# B&R Automation Studio project CombinedLinenSoiledA9KAN (part 18)

#### _actIFCmd.st
```iecst
(********************************************************************
 * COPYRIGHT -- Herbert Kannegiesser GmbH
 ********************************************************************
 * Program: svCPCache
 * File: _actIFCmd.st
 * Author: hunholz
 * Created: March 30, 2012
 ********************************************************************
 * Implementation of program svCPCache
 ********************************************************************)

(* Add a new action to your IEC program or library *)
ACTION _actIFCmd:

	CASE _enCmd OF

		cs_CmdIdle:

		// Warte auf Kommando

			CASE IFsvCPCache.In.wCmd OF

				KG_CMD_NOCOMMAND:

					IFsvCPCache.Out.wCmdResponse := KG_CMD_NOCOMMAND;

				SVCPCACHE_CMD_GETPROG:

					IFsvCPCache.Out.rRespSoilFactor 		:= 1.0;
					IFsvCPCache.Out.utfRespCategoryName		:= "";
					IFsvCPCache.Out.wRespColidxBack			:= 15;
					IFsvCPCache.Out.wRespColidxFor			:= 1;
					IFsvCPCache.Out.wRespLoadrate			:= 100;
					IFsvCPCache.Out.wRespProgramNo			:= 0;
					IFsvCPCache.Out.utfRespProgramName		:= "";

					IFsvCPCache.Out.wRespFromDB				:= SVCPCACHE_DBREQ_LOCAL;

					_TrimCat(sCategory := IFsvCPCache.In.sReqCategory);
					_sCategory := _TrimCat.sOutCategory;

					IF _sCategory <> '' THEN

						// Suche Kategorie auf jeden Fall lokal

						_xCategoryExist := FALSE;
						_wCategoryIdx := 0;

						FOR _i := 1 TO SVCPCACHE_CNT_RELATIONS DO

							IF _CPCache[_i].dtTimeStamp = USINT_TO_DT(0) THEN
								EXIT;
							ELSIF _CPCache[_i].sCategory = _sCategory THEN
								_xCategoryExist := TRUE;
								_wCategoryIdx := _i;
								EXIT;
							END_IF

						END_FOR

						// Entscheidung, ob in der Datenbank gesucht werden soll

						IF IFsvCPCache.In.wReqUseDB = SVCPCACHE_DBREQ_LOCAL THEN

							IF _xCategoryExist THEN

								IFsvCPCache.Out.rRespSoilFactor 		:= _CPCache[_wCategoryIdx].rSoilfactor;
								IFsvCPCache.Out.utfRespCategoryName		:= _CPCache[_wCategoryIdx].utfCategoryName;
								IFsvCPCache.Out.wRespColidxBack			:= _CPCache[_wCategoryIdx].wColBack;
								IFsvCPCache.Out.wRespColidxFor			:= _CPCache[_wCategoryIdx].wColFor;
								IFsvCPCache.Out.wRespLoadrate			:= _CPCache[_wCategoryIdx].wLoadrate;
								IFsvCPCache.Out.wRespProgramNo			:= _CPCache[_wCategoryIdx].wProgramNo;

								FOR _i := 1 TO IFmnParam.Out.Edit.wCntNamelist DO

									IF IFmnParam.Out.Edit.wNameListNo[_i] = IFsvCPCache.Out.wRespProgramNo THEN
										IFsvCPCache.Out.utfRespProgramName := IFmnParam.Out.Edit.utfNameListName[_i];
										EXIT;
									END_IF

								END_FOR

								IFsvCPCache.Out.wCmdResponse := SVCPCACHE_CMD_GETPROG;
								_enCmd := cs_CmdWaitForNoCommand;

							ELSE

								IFsvCPCache.Out.wCmdResponse := SVCPCACHE_STAT_CATEGORYNOTEXIST;
								_enCmd := cs_CmdWaitForNoCommand;

							END_IF

						ELSE // Abfrage der Datenbank starten

							IF IFhlDFII.Out.xConnected THEN

								IFsvCPCache.Out.wCmdResponse := KG_STAT_BUSY;
								_enCmd := cs_CmdWaitForDB;

							ELSE

								IFsvCPCache.Out.wCmdResponse := SVCPCACHE_STAT_DBNOTREADY;
								_enCmd := cs_CmdWaitForNoCommand;

								IF _xCategoryExist THEN

									IFsvCPCache.Out.rRespSoilFactor 		:= _CPCache[_wCategoryIdx].rSoilfactor;
									IFsvCPCache.Out.utfRespCategoryName		:= _CPCache[_wCategoryIdx].utfCategoryName;
									IFsvCPCache.Out.wRespColidxBack			:= _CPCache[_wCategoryIdx].wColBack;
									IFsvCPCache.Out.wRespColidxFor			:= _CPCache[_wCategoryIdx].wColFor;
									IFsvCPCache.Out.wRespLoadrate			:= _CPCache[_wCategoryIdx].wLoadrate;
									IFsvCPCache.Out.wRespProgramNo			:= _CPCache[_wCategoryIdx].wProgramNo;

									FOR _i := 1 TO IFmnParam.Out.Edit.wCntNamelist DO

										IF IFmnParam.Out.Edit.wNameListNo[_i] = IFsvCPCache.Out.wRespProgramNo THEN
											IFsvCPCache.Out.utfRespProgramName := IFmnParam.Out.Edit.utfNameListName[_i];
											EXIT;
										END_IF

									END_FOR

								END_IF

							END_IF

						END_IF

					ELSE

						IFsvCPCache.Out.wCmdResponse := SVCPCACHE_STAT_INVALIDCATEGORY;
						_enCmd := cs_CmdWaitForNoCommand;

					END_IF

				SVCPCACHE_CMD_INSERTCATEGORY:

					_wCmd := SVCPCACHE_CMD_INSERTCATEGORY;

					IF IFsvCPCache.Out.wCntRelations < SVCPCACHE_CNT_RELATIONS THEN

						_TrimCat(sCategory := IFsvCPCache.In.sReqCategory);
						_sCategory := _TrimCat.sOutCategory;

						IF _sCategory <> '' THEN

							_xCategoryExist := FALSE;

							FOR _i := 1 TO SVCPCACHE_CNT_RELATIONS DO

								IF _CPCache[_i].dtTimeStamp = USINT_TO_DT(0) THEN
									EXIT;
								ELSIF _CPCache[_i].sCategory = _sCategory THEN
									_xCategoryExist := TRUE;
									EXIT;
								END_IF

							END_FOR

							IF NOT _xCategoryExist THEN

								_DTGetTime(enable := TRUE);

								FOR _i := 1 TO SVCPCACHE_CNT_RELATIONS DO

									IF _CPCache[_i].dtTimeStamp = USINT_TO_DT(0) THEN

										_CPCache[_i].dtTimeStamp := _DTGetTime.DT1;
										_CPCache[_i].sCategory := _sCategory;
										_CPCache[_i].utfCategoryName := IFsvCPCache.In.utfReqCategoryName;
										_CPCache[_i].wProgramNo := IFsvCPCache.In.wReqProgramNo;
										_CPCache[_i].rSoilfactor := IFsvCPCache.In.rReqSoilfactor;
										_CPCache[_i].wLoadrate := IFsvCPCache.In.wReqLoadrate;
										_CPCache[_i].wColFor := IFsvCPCache.In.wReqColidxFor;
										_CPCache[_i].wColBack := IFsvCPCache.In.wReqColidxBack;

										IFsvCPCache.Out.wCntRelations := IFsvCPCache.Out.wCntRelations + 1;

										EXIT;

									ELSIF brsstrcmp(ADR(_CPCache[_i].sCategory),ADR(_sCategory)) > 0 THEN

										brsmemmove(ADR(_CPCache[_i+1]), ADR(_CPCache[_i]), SIZEOF(_CPCache[1])*(IFsvCPCache.Out.wCntRelations-_i+1) );

										_CPCache[_i].dtTimeStamp := _DTGetTime.DT1;
										_CPCache[_i].sCategory := _sCategory;
										_CPCache[_i].utfCategoryName := IFsvCPCache.In.utfReqCategoryName;
										_CPCache[_i].wProgramNo := IFsvCPCache.In.wReqProgramNo;
										_CPCache[_i].rSoilfactor := IFsvCPCache.In.rReqSoilfactor;
										_CPCache[_i].wLoadrate := IFsvCPCache.In.wReqLoadrate;
										_CPCache[_i].wColFor := IFsvCPCache.In.wReqColidxFor;
										_CPCache[_i].wColBack := IFsvCPCache.In.wReqColidxBack;

										IFsvCPCache.Out.wCntRelations := IFsvCPCache.Out.wCntRelations + 1;

										EXIT;

									END_IF

								END_FOR

								_enSave := cs_SaveCreateCSV;

								_enCmd := cs_CmdSave;

							ELSE

								IFsvCPCache.Out.wCmdResponse := SVCPCACHE_STAT_CATEGORYEXIST;
								_enCmd := cs_CmdWaitForNoCommand;

							END_IF

						ELSE

							IFsvCPCache.Out.wCmdResponse := SVCPCACHE_STAT_INVALIDCATEGORY;
							_enCmd := cs_CmdWaitForNoCommand;

						END_IF

					ELSE

						IFsvCPCache.Out.wCmdResponse := SVCPCACHE_STAT_NOSPACE;
						_enCmd := cs_CmdWaitForNoCommand;

					END_IF

				SVCPCACHE_CMD_UPDATECATEGORY:

					_wCmd := SVCPCACHE_CMD_UPDATECATEGORY;

					IF IFsvCPCache.Out.wCntRelations > 0 THEN

						_TrimCat(sCategory := IFsvCPCache.In.sReqCategory);
						_sCategory := _TrimCat.sOutCategory;

						IF _sCategory <> '' THEN

							_xCategoryExist := FALSE;

							FOR _i := 1 TO SVCPCACHE_CNT_RELATIONS DO

								IF _CPCache[_i].dtTimeStamp = USINT_TO_DT(0) THEN
									EXIT;
								ELSIF _CPCache[_i].sCategory = _sCategory THEN
									_xCategoryExist := TRUE;
									EXIT;
								END_IF

							END_FOR

							IF _xCategoryExist THEN

								_DTGetTime(enable := TRUE);

								_CPCache[_i].dtTimeStamp := _DTGetTime.DT1;
								_CPCache[_i].sCategory := _sCategory;
								_CPCache[_i].utfCategoryName := IFsvCPCache.In.utfReqCategoryName;
								_CPCache[_i].wProgramNo := IFsvCPCache.In.wReqProgramNo;
								_CPCache[_i].rSoilfactor := IFsvCPCache.In.rReqSoilfactor;
								_CPCache[_i].wLoadrate := IFsvCPCache.In.wReqLoadrate;
								_CPCache[_i].wColFor := IFsvCPCache.In.wReqColidxFor;
								_CPCache[_i].wColBack := IFsvCPCache.In.wReqColidxBack;

								_enSave := cs_SaveCreateCSV;

								_enCmd := cs_CmdSave;

							ELSE

								IFsvCPCache.Out.wCmdResponse := SVCPCACHE_STAT_CATEGORYNOTEXIST;
								_enCmd := cs_CmdWaitForNoCommand;

							END_IF

						ELSE

							IFsvCPCache.Out.wCmdResponse := SVCPCACHE_STAT_INVALIDCATEGORY;
							_enCmd := cs_CmdWaitForNoCommand;

						END_IF

					ELSE

						IFsvCPCache.Out.wCmdResponse := SVCPCACHE_STAT_CATEGORYLISTEMPTY;
						_enCmd := cs_CmdWaitForNoCommand;

					END_IF

				SVCPCACHE_CMD_DELETECATEGORY:

					_wCmd := SVCPCACHE_CMD_DELETECATEGORY;

					IF IFsvCPCache.Out.wCntRelations > 0 THEN

						_TrimCat(sCategory := IFsvCPCache.In.sReqCategory);
						_sCategory := _TrimCat.sOutCategory;

						IF _sCategory <> '' THEN

							_xCategoryExist := FALSE;

							FOR _i := 1 TO SVCPCACHE_CNT_RELATIONS DO

								IF _CPCache[_i].dtTimeStamp = USINT_TO_DT(0) THEN
									EXIT;
								ELSIF _CPCache[_i].sCategory = _sCategory THEN
									_xCategoryExist := TRUE;
									EXIT;
								END_IF

							END_FOR

							IF _xCategoryExist THEN

								IF _i < IFsvCPCache.Out.wCntRelations THEN

									brsmemmove(ADR(_CPCache[_i]), ADR(_CPCache[_i+1]), SIZEOF(_CPCache[1])*(IFsvCPCache.Out.wCntRelations-_i) );

								END_IF

								brsmemset(ADR(_CPCache[IFsvCPCache.Out.wCntRelations]), 0, SIZEOF(_CPCache[1]));

								IFsvCPCache.Out.wCntRelations := IFsvCPCache.Out.wCntRelations - 1;

								_enSave := cs_SaveCreateCSV;

								_enCmd := cs_CmdSave;

							ELSE

								IFsvCPCache.Out.wCmdResponse := SVCPCACHE_STAT_CATEGORYNOTEXIST;
								_enCmd := cs_CmdWaitForNoCommand;

							END_IF

						ELSE

							IFsvCPCache.Out.wCmdResponse := SVCPCACHE_STAT_INVALIDCATEGORY;
							_enCmd := cs_CmdWaitForNoCommand;

						END_IF

					ELSE

						IFsvCPCache.Out.wCmdResponse := SVCPCACHE_STAT_CATEGORYLISTEMPTY;
						_enCmd := cs_CmdWaitForNoCommand;

					END_IF

				SVCPCACHE_CMD_SETOFFSET:

					IFsvCPCache.Out.wListOffset := IFsvCPCache.In.wSetOffset;
					_actFillCPList;

					IFsvCPCache.Out.wCmdResponse := SVCPCACHE_CMD_SETOFFSET;
					_enCmd := cs_CmdWaitForNoCommand;

				ELSE

					IFsvCPCache.Out.wCmdResponse := KG_CMDSTAT_NOTVALID;
					_enCmd := cs_CmdWaitForNoCommand;

			END_CASE

		cs_CmdSave:

			IF _enSave = cs_SaveRdySuccess THEN

				_actFillCPList;

				IFsvCPCache.Out.wCmdResponse := _wCmd;
				_enCmd := cs_CmdWaitForNoCommand;

			ELSIF _enSave = cs_SaveRdyFault THEN

				IFsvCPCache.Out.wCmdResponse := _wSaveCSVstatus;
				_enCmd := cs_CmdWaitForNoCommand;

			END_IF

		cs_CmdWaitForDB:

			IF IFhlDFII.In.ReqProgByCat.wRequest = 0 AND IFhlDFII.Out.RespProgByCat.wResponse = 0 THEN

				IFhlDFII.In.ReqProgByCat.sCategoryNo_In := IFsvCPCache.In.sReqCategory;
				IFhlDFII.In.ReqProgByCat.wRequest		:= 2;

			ELSIF IFhlDFII.In.ReqProgByCat.wRequest = 2 AND IFhlDFII.Out.RespProgByCat.wResponse = 2 THEN

				_DTGetTime(enable := TRUE);

				IFsvCPCache.Out.rRespSoilFactor 		:= IFhlDFII.Out.RespProgByCat.rSoilfactor;
				IFsvCPCache.Out.utfRespCategoryName 	:= STRING_TO_WSTRING(IFhlDFII.Out.RespProgByCat.sCategoryName);
				IFsvCPCache.Out.wRespColidxBack			:= IFhlDFII.Out.RespProgByCat.wColorIdxBack;
				IFsvCPCache.Out.wRespColidxFor			:= IFhlDFII.Out.RespProgByCat.wColorIdxFor;
				IFsvCPCache.Out.wRespLoadrate			:= IFhlDFII.Out.RespProgByCat.wLoadrate;
				IFsvCPCache.Out.wRespProgramNo			:= IFhlDFII.Out.RespProgByCat.bProgramNo;

				FOR _i := 1 TO IFmnParam.Out.Edit.wCntNamelist DO

					IF IFmnParam.Out.Edit.wNameListNo[_i] = IFsvCPCache.Out.wRespProgramNo THEN
						IFsvCPCache.Out.utfRespProgramName := IFmnParam.Out.Edit.utfNameListName[_i];
						EXIT;
					END_IF

				END_FOR

				IFsvCPCache.Out.wRespFromDB				:= SVCPCACHE_DBREQ_DFII;

				IF _xCategoryExist AND
					_CPCache[_wCategoryIdx].utfCategoryName = IFsvCPCache.Out.utfRespCategoryName AND
					_CPCache[_wCategoryIdx].rSoilfactor = IFsvCPCache.Out.rRespSoilFactor AND
					_CPCache[_wCategoryIdx].wLoadrate = IFsvCPCache.Out.wRespLoadrate AND
					_CPCache[_wCategoryIdx].wColBack = IFsvCPCache.Out.wRespColidxBack AND
					_CPCache[_wCategoryIdx].wColFor = IFsvCPCache.Out.wRespColidxFor AND
					_CPCache[_wCategoryIdx].wProgramNo =  IFsvCPCache.Out.wRespProgramNo THEN

					// Lokale Daten sind gleich den Daten aus der Datenbank

					IFsvCPCache.Out.wCmdResponse			:= SVCPCACHE_CMD_GETPROG;
					_enCmd := cs_CmdWaitForNoCommand;

				ELSIF _xCategoryExist THEN

					// Lokale Daten werden aktualisiert

					_CPCache[_wCategoryIdx].utfCategoryName := STRING_TO_WSTRING(IFhlDFII.Out.RespProgByCat.sCategoryName);
					_CPCache[_wCategoryIdx].rSoilfactor 	:= IFhlDFII.Out.RespProgByCat.rSoilfactor;
					_CPCache[_wCategoryIdx].wLoadrate 		:= IFhlDFII.Out.RespProgByCat.wLoadrate;
					_CPCache[_wCategoryIdx].wColBack 		:= IFhlDFII.Out.RespProgByCat.wColorIdxBack;
					_CPCache[_wCategoryIdx].wColFor 		:= IFhlDFII.Out.RespProgByCat.wColorIdxFor;
					_CPCache[_wCategoryIdx].wProgramNo 		:= IFhlDFII.Out.RespProgByCat.bProgramNo;
					_CPCache[_wCategoryIdx].dtTimeStamp		:= _DTGetTime.DT1;

					_wCmd := SVCPCACHE_CMD_GETPROG;
					_enSave := cs_SaveCreateCSV;
					_enCmd := cs_CmdSave;

				ELSE

					// Es wird versucht eine neue Kategorie in den lokalen Speicher abzulegen

					IF IFsvCPCache.Out.wCntRelations < SVCPCACHE_CNT_RELATIONS THEN

						FOR _i := 1 TO SVCPCACHE_CNT_RELATIONS DO

							IF _CPCache[_i].dtTimeStamp = USINT_TO_DT(0) THEN

								_CPCache[_i].dtTimeStamp 		:= _DTGetTime.DT1;
								_CPCache[_i].sCategory 			:= _sCategory;
								_CPCache[_i].utfCategoryName 	:= STRING_TO_WSTRING(IFhlDFII.Out.RespProgByCat.sCategoryName);
								_CPCache[_i].wProgramNo 		:= IFhlDFII.Out.RespProgByCat.bProgramNo;
								_CPCache[_i].rSoilfactor 		:= IFhlDFII.Out.RespProgByCat.rSoilfactor;
								_CPCache[_i].wLoadrate 			:= IFhlDFII.Out.RespProgByCat.wLoadrate;
								_CPCache[_i].wColFor 			:= IFhlDFII.Out.RespProgByCat.wColorIdxFor;
								_CPCache[_i].wColBack 			:= IFhlDFII.Out.RespProgByCat.wColorIdxBack;

								IFsvCPCache.Out.wCntRelations := IFsvCPCache.Out.wCntRelations + 1;

								EXIT;

							ELSIF brsstrcmp(ADR(_CPCache[_i].sCategory),ADR(_sCategory)) > 0 THEN

								brsmemmove(ADR(_CPCache[_i+1]), ADR(_CPCache[_i]), SIZEOF(_CPCache[1])*(IFsvCPCache.Out.wCntRelations-_i+1) );

								_CPCache[_i].dtTimeStamp 		:= _DTGetTime.DT1;
								_CPCache[_i].sCategory 			:= _sCategory;
								_CPCache[_i].utfCategoryName 	:= STRING_TO_WSTRING(IFhlDFII.Out.RespProgByCat.sCategoryName);
								_CPCache[_i].wProgramNo 		:= IFhlDFII.Out.RespProgByCat.bProgramNo;
								_CPCache[_i].rSoilfactor 		:= IFhlDFII.Out.RespProgByCat.rSoilfactor;
								_CPCache[_i].wLoadrate 			:= IFhlDFII.Out.RespProgByCat.wLoadrate;
								_CPCache[_i].wColFor 			:= IFhlDFII.Out.RespProgByCat.wColorIdxFor;
								_CPCache[_i].wColBack 			:= IFhlDFII.Out.RespProgByCat.wColorIdxBack;

								IFsvCPCache.Out.wCntRelations := IFsvCPCache.Out.wCntRelations + 1;

								EXIT;

							END_IF

						END_FOR

						_wCmd := SVCPCACHE_CMD_GETPROG;
						_enSave := cs_SaveCreateCSV;
						_enCmd := cs_CmdSave;

					ELSE

						// Kein Platz für eine neue Kategorie

						IFsvCPCache.Out.wCmdResponse			:= SVCPCACHE_CMD_GETPROG;
						_enCmd := cs_CmdWaitForNoCommand;

					END_IF

				END_IF

				IFhlDFII.In.ReqProgByCat.wRequest		:= 0;

			ELSIF IFhlDFII.In.ReqProgByCat.wRequest = 2 AND IFhlDFII.Out.RespProgByCat.wResponse <> 65535 AND IFhlDFII.Out.RespProgByCat.wResponse <> 0 THEN

				IF _xCategoryExist THEN

					IFsvCPCache.Out.rRespSoilFactor 		:= _CPCache[_wCategoryIdx].rSoilfactor;
					IFsvCPCache.Out.utfRespCategoryName		:= _CPCache[_wCategoryIdx].utfCategoryName;
					IFsvCPCache.Out.wRespColidxBack			:= _CPCache[_wCategoryIdx].wColBack;
					IFsvCPCache.Out.wRespColidxFor			:= _CPCache[_wCategoryIdx].wColFor;
					IFsvCPCache.Out.wRespLoadrate			:= _CPCache[_wCategoryIdx].wLoadrate;
					IFsvCPCache.Out.wRespProgramNo			:= _CPCache[_wCategoryIdx].wProgramNo;

					FOR _i := 1 TO IFmnParam.Out.Edit.wCntNamelist DO

						IF IFmnParam.Out.Edit.wNameListNo[_i] = IFsvCPCache.Out.wRespProgramNo THEN
							IFsvCPCache.Out.utfRespProgramName := IFmnParam.Out.Edit.utfNameListName[_i];
							EXIT;
						END_IF

					END_FOR

					IFsvCPCache.Out.wCmdResponse 			:= SVCPCACHE_CMD_GETPROG;

				ELSE

					IFsvCPCache.Out.wCmdResponse			:= IFhlDFII.Out.RespProgByCat.wResponse;

				END_IF

				IFhlDFII.In.ReqProgByCat.wRequest		:= 0;
				_enCmd := cs_CmdWaitForNoCommand;

			END_IF

		cs_CmdWaitForNoCommand:

			IF IFsvCPCache.In.wCmd = KG_CMD_NOCOMMAND THEN

				IFsvCPCache.Out.wCmdResponse := KG_STAT_OK;

				_enCmd := cs_CmdIdle;

			END_IF

	END_CASE

END_ACTION
```

#### _actSaveCSV.st
```iecst
(********************************************************************
 * COPYRIGHT -- Herbert Kannegiesser GmbH
 ********************************************************************
 * Program: svCPCache
 * File: _actSaveCSV.st
 * Author: hunholz
 * Created: March 30, 2012
 ********************************************************************
 * Implementation of program svCPCache
 ********************************************************************)

(* Schrittkette zum Speichern der Kategorie-Programm-Zuordnung *)
ACTION _actSaveCSV:

	_wSaveCSVstatus := ERR_OK;

	CASE _enSave OF

		cs_SaveIdle:

			// Tue nichts

		cs_SaveCreateCSV:

			_SaveMemPartAlloc(enable := TRUE, ident := _MemPartCreate.ident , len := _lMemLen);
			_lWriteSize := 0;

			IF _SaveMemPartAlloc.status = ERR_OK THEN

				_WriteBOM(enable := TRUE, pMem := _SaveMemPartAlloc.mem, lMaxSize := _lMemLen, lSize := _lWriteSize);

				// Kopfdaten schreiben
				_WriteComment(enable := TRUE, pMem := _SaveMemPartAlloc.mem, lMaxSize := _lMemLen, sComment := CONCAT('svCPCache Version: ',svCPCacheStatAd.sPkgVersion) , lSize := _lWriteSize);
				_WriteNewLine(enable := TRUE, pMem := _SaveMemPartAlloc.mem, lMaxSize := _lMemLen, lSize := _lWriteSize);

				_MachineNoRow.utfMachineNo := IFmnParam.Out.utfMachineNumber;
				_WriteMachineNo(enable := TRUE, pMem := _SaveMemPartAlloc.mem, lMaxSize := _lMemLen, MachineNoRow := _MachineNoRow, lSize := _lWriteSize);

				_WriteNewLine(enable := TRUE, pMem := _SaveMemPartAlloc.mem, lMaxSize := _lMemLen, lSize := _lWriteSize);

				_DTGetTime(enable := TRUE);
				_HeaderTimeRow.dtTimestamp := _DTGetTime.DT1;

				_WriteTimeStamp(enable := TRUE, pMem := _SaveMemPartAlloc.mem, lMaxSize := _lMemLen, TimeRow := _HeaderTimeRow, lSize := _lWriteSize);

				_WriteNewLine(enable := TRUE, pMem := _SaveMemPartAlloc.mem, lMaxSize := _lMemLen, lSize := _lWriteSize);

				FOR _sci := 1 TO SVCPCACHE_CNT_RELATIONS DO

					IF _CPCache[_sci].dtTimeStamp <> USINT_TO_DT(0) AND _CPCache[_sci].sCategory <> '' THEN

						_WriteCP(enable := TRUE, pMem := _SaveMemPartAlloc.mem, lMaxSize := _lMemLen, CPRow := _CPCache[_sci], lSize := _lWriteSize);

					END_IF

				END_FOR

				_enSave := cs_SaveDeleteFile;

			ELSE

				_wSaveCSVstatus := SVCPCACHE_STAT_MEMALLOC;
				_enSave := cs_SaveRdyFault;

			END_IF

		cs_SaveDeleteFile:

			_FileDelete(enable := TRUE, pDevice := ADR(KG_DEVICE_COMPACTFLASH), pName := ADR(_SVCPCACHE_CSV_FILE));

			IF _FileDelete.status <> ERR_FUB_BUSY THEN

				_enSave := cs_SaveCreateFile;

			END_IF

		//==============================================
		// Exportdatei erzeugen
		//==============================================
		cs_SaveCreateFile:

			_FileCreate(enable := TRUE, pDevice := ADR(KG_DEVICE_COMPACTFLASH), pFile := ADR(_SVCPCACHE_CSV_FILE) );

			IF _FileCreate.status = ERR_OK THEN

				_enSave := cs_SaveOpenFile;

			ELSIF _FileCreate.status <> ERR_FUB_BUSY THEN

				_SaveMemPartFree(enable := TRUE, ident := _MemPartCreate.ident, mem := _SaveMemPartAlloc.mem);

				_wSaveCSVstatus := SVCPCACHE_STAT_CREATEFILE;
				_enSave := cs_SaveRdyFault;

			END_IF

		//==============================================
		// Exportdatei öffnen
		//==============================================
		cs_SaveOpenFile:

			_FileOpen(enable := TRUE, pDevice := ADR(KG_DEVICE_COMPACTFLASH), pFile := ADR(_SVCPCACHE_CSV_FILE), mode := fiWRITE_ONLY);

			IF _FileOpen.status = ERR_OK THEN

				_enSave := cs_SaveWriteFile;

			ELSIF _FileOpen.status <> ERR_FUB_BUSY THEN

				_SaveMemPartFree(enable := TRUE, ident := _MemPartCreate.ident, mem := _SaveMemPartAlloc.mem);

				_wSaveCSVstatus := SVCPCACHE_STAT_OPENFILE;
				_enSave := cs_SaveRdyFault;

			END_IF

		//==============================================
		// Exportdatei schreiben
		//==============================================
		cs_SaveWriteFile:

			_FileWrite(enable := TRUE, ident := _FileOpen.ident, offset := 0, pSrc :=_SaveMemPartAlloc.mem, len := _lWriteSize);

			IF _FileWrite.status = ERR_OK THEN

				_SaveMemPartFree(enable := TRUE, ident := _MemPartCreate.ident, mem := _SaveMemPartAlloc.mem);
				_enSave := cs_SaveCloseFile;

			ELSIF _FileWrite.status <> ERR_FUB_BUSY THEN

				_SaveMemPartFree(enable := TRUE, ident := _MemPartCreate.ident, mem := _SaveMemPartAlloc.mem);

				_wSaveCSVstatus := SVCPCACHE_STAT_WRITEFILE;
				_enSave := cs_SaveCloseFile;

			END_IF

		//==============================================
		// Exportdatei schließen
		//==============================================
		cs_SaveCloseFile:

			_FileClose(enable := TRUE, ident := _FileOpen.ident);

			IF _FileClose.status <> ERR_FUB_BUSY THEN

				IF _wSaveCSVstatus = ERR_OK THEN

					_enSave := cs_SaveRdySuccess;

				ELSE

					_enSave := cs_SaveRdyFault;

				END_IF

			END_IF

		cs_SaveRdyFault:

			// Mit Fehler beendet

		cs_SaveRdySuccess:

			// Erfolgreich beendet

	END_CASE

END_ACTION
```

#### _TrimCategory.st - Entfernt führende Nullen und Leerzeichen, sowie folgende Leerzeichen
```iecst
(********************************************************************
 * COPYRIGHT -- Herbert Kannegiesser GmbH
 ********************************************************************
 * Program: svCPCache
 * File: _TrimCategory.st
 * Author: hunholz
 * Created: March 30, 2012
 ********************************************************************
 * Implementation of program svCPCache
 ********************************************************************)

(* Entfernt führende Nullen und Leerzeichen, sowie folgende Leerzeichen *)
FUNCTION_BLOCK _TrimCategory

	sOutCategory := sCategory;

	IF LEN(sOutCategory) > 0 THEN
		REPEAT
			_iFound := FIND(sOutCategory,' ');

			IF _iFound <> 0 THEN
				sOutCategory := DELETE(sOutCategory,1,_iFound);
			END_IF

			UNTIL
			_iFound = 0 OR LEN(sOutCategory) = 0
		END_REPEAT
	END_IF

	IF LEN(sOutCategory) > 0 THEN
		REPEAT
			_iFound := FIND(sOutCategory,'0');

			IF _iFound = 1 THEN
				sOutCategory := DELETE(sOutCategory,1,_iFound);
			END_IF

			UNTIL
			_iFound <> 1 OR LEN(sOutCategory) = 0
		END_REPEAT
	END_IF

END_FUNCTION_BLOCK
```

### Package Logical/Mewa/KGFrameworkShare - Benutzereinstellungen

### hlDFII.Glob.var - Package variables
```iecst
(********************************************************************
 * COPYRIGHT -- Herbert Kannegiesser GmbH
 ********************************************************************
 * File: hlDFII.Glob.var
 * Author: hunholz
 * Created: January 12, 2012
 ********************************************************************
 * Global variables of project POWERTRANSplus
 ********************************************************************)
VAR CONSTANT
	HLDFII_RUN_CLIENT : BOOL := TRUE;
	HLDFII_IDX_CPCACHE_MAX : UINT := 99;
	HLDFII_UDP_PORT_LOG4NET : UINT := 1009;
END_VAR
```

### mnSystemGlob.var - Package variables
```iecst
(********************************************************************
 * COPYRIGHT -- Herbert Kannegiesser GmbH
 ********************************************************************
 * File: mnSystemGlob.var
 * Author: hunholz
 * Created: Mar 16, 2012
 ********************************************************************
 * Global variables of project KGFramework
 ********************************************************************)
VAR CONSTANT
	MNSYSTEM_IDX_KGMSGSTAT : UINT := 102;
END_VAR
```


### Package Logical/Mewa/KGFrameworkShare/Pkg_mnMsgShare - Konfiguration des mnMsg

### Data object Logical/Mewa/KGFrameworkShare/Pkg_mnMsgShare/CfgMsgStat (Simple) - Configuration of Messagestatistics

#### CfgMsgStat.dat
```
(********************************************************************
 * COPYRIGHT -- Microsoft
 ********************************************************************
 * Data object: CfgMsgStat
 * File: CfgMsgStat.dat
 * Author: hunholz / Subramaniam
 * Created: January 05, 2011
 * Changed : December 21, 2011
 ********************************************************************
 * Data object file: CfgMsgStat.dat
 ********************************************************************)
; Configurationlist for Messagemanager

00002; Versionnumber
;*****************************************************************

; Configurationlist
;--------------------------
; Function_ID, Message_No, Instance, Reserve
; ****************************
; Erste Funktionsgruppe
;*****************************
;    +---------------------------------------------- Function_ID
;    | 		  +------------------------------------ Message_No
;    |        |		+------------------------- Instance
;    |        |		|		 +--------------- Reserve
;    |		  |		|		 |
;****************************
; Parameter Manager
;*****************************
00001, 00001, 00000, 00000;
00001, 00002, 00000, 00000;
00001, 00009, 00000, 00000;
00001, 20000, 00000, 00000;
;****************************
; Meldungsmanager mnMsg
;*****************************
00002, 01000, 00000, 00000;
00002, 01003, 00000, 00000;
; ****************************
; Dritte Funktionsgruppe
;*****************************
00004, 00010, 00000, 00000;
00004, 00011, 00000, 00000;
00004, 00012, 00000, 00000;
00004, 00013, 00000, 00000;
00004, 20000, 00000, 00000;
00004, 20001, 00000, 00000;
00004, 20002, 00000, 00000;
; ****************************
; mnMaster
;*****************************
00101, 00200, 00000, 00000;
00101, 00201, 00000, 00000;
00101, 01001, 00000, 00000;
; ****************************
; mnLoad
;*****************************
00102, 00001, 00000, 00000;
00102, 00002, 00000, 00000;
00102, 00003, 00000, 00000;
00102, 00004, 00000, 00000;
00102, 00005, 00000, 00000;
00102, 00006, 00000, 00000;
00102, 00007, 00000, 00000;
00102, 00011, 00000, 00000;
00102, 00012, 00000, 00000;
; ****************************
; mnUnload
;*****************************
00103, 00001, 00000, 00000;
00103, 00007, 00000, 00000;
; ****************************
; mnComp
;*****************************
00104, 00100, 00001, 00000;
00104, 00100, 00002, 00000;
00104, 00100, 00003, 00000;
00104, 00100, 00004, 00000;
00104, 00100, 00005, 00000;
00104, 00100, 00006, 00000;
00104, 00100, 00007, 00000;
00104, 00100, 00008, 00000;
00104, 00100, 00009, 00000;
00104, 00100, 00010, 00000;
00104, 00100, 00011, 00000;
00104, 00100, 00012, 00000;
00104, 00100, 00013, 00000;
00104, 00100, 00014, 00000;
00104, 00100, 00015, 00000;
00104, 00100, 00016, 00000;
00104, 00100, 00017, 00000;
00104, 00100, 00018, 00000;
00104, 00100, 00019, 00000;
00104, 00100, 00020, 00000;
00104, 00100, 00021, 00000;
00104, 00100, 00022, 00000;
00104, 00100, 00023, 00000;
00104, 00100, 00024, 00000;
00104, 00100, 00025, 00000;
00104, 00100, 00026, 00000;
00104, 00100, 00027, 00000;
00104, 00100, 00028, 00000;
00104, 00100, 00029, 00000;
00104, 00100, 00030, 00000;
00104, 00101, 00001, 00000;
00104, 00101, 00002, 00000;
00104, 00101, 00003, 00000;
00104, 00101, 00004, 00000;
00104, 00101, 00005, 00000;
00104, 00101, 00006, 00000;
00104, 00101, 00007, 00000;
00104, 00101, 00008, 00000;
00104, 00101, 00009, 00000;
00104, 00101, 00010, 00000;
00104, 00101, 00011, 00000;
00104, 00101, 00012, 00000;
00104, 00101, 00013, 00000;
00104, 00101, 00014, 00000;
00104, 00101, 00015, 00000;
00104, 00101, 00016, 00000;
00104, 00101, 00017, 00000;
00104, 00101, 00018, 00000;
00104, 00101, 00019, 00000;
00104, 00101, 00020, 00000;
00104, 00101, 00021, 00000;
00104, 00101, 00022, 00000;
00104, 00101, 00023, 00000;
00104, 00101, 00024, 00000;
00104, 00101, 00025, 00000;
00104, 00101, 00026, 00000;
00104, 00101, 00027, 00000;
00104, 00101, 00028, 00000;
00104, 00101, 00029, 00000;
00104, 00101, 00030, 00000;
00104, 00102, 00001, 00000;
00104, 00102, 00002, 00000;
00104, 00102, 00003, 00000;
00104, 00102, 00004, 00000;
00104, 00102, 00005, 00000;
00104, 00102, 00006, 00000;
00104, 00102, 00007, 00000;
00104, 00102, 00008, 00000;
00104, 00102, 00009, 00000;
00104, 00102, 00010, 00000;
00104, 00102, 00011, 00000;
00104, 00102, 00012, 00000;
00104, 00102, 00013, 00000;
00104, 00102, 00014, 00000;
00104, 00102, 00015, 00000;
00104, 00102, 00016, 00000;
00104, 00102, 00017, 00000;
00104, 00102, 00018, 00000;
00104, 00102, 00019, 00000;
00104, 00102, 00020, 00000;
00104, 00102, 00021, 00000;
00104, 00102, 00022, 00000;
00104, 00102, 00023, 00000;
00104, 00102, 00024, 00000;
00104, 00102, 00025, 00000;
00104, 00102, 00026, 00000;
00104, 00102, 00027, 00000;
00104, 00102, 00028, 00000;
00104, 00102, 00029, 00000;
00104, 00102, 00030, 00000;
00104, 00103, 00001, 00000;
00104, 00103, 00002, 00000;
00104, 00103, 00003, 00000;
00104, 00103, 00004, 00000;
00104, 00103, 00005, 00000;
00104, 00103, 00006, 00000;
00104, 00103, 00007, 00000;
00104, 00103, 00008, 00000;
00104, 00103, 00009, 00000;
00104, 00103, 00010, 00000;
00104, 00103, 00011, 00000;
00104, 00103, 00012, 00000;
00104, 00103, 00013, 00000;
00104, 00103, 00014, 00000;
00104, 00103, 00015, 00000;
00104, 00103, 00016, 00000;
00104, 00103, 00017, 00000;
00104, 00103, 00018, 00000;
00104, 00103, 00019, 00000;
00104, 00103, 00020, 00000;
00104, 00103, 00021, 00000;
00104, 00103, 00022, 00000;
00104, 00103, 00023, 00000;
00104, 00103, 00024, 00000;
00104, 00103, 00025, 00000;
00104, 00103, 00026, 00000;
00104, 00103, 00027, 00000;
00104, 00103, 00028, 00000;
00104, 00103, 00029, 00000;
00104, 00103, 00030, 00000;
00104, 00110, 00001, 00000;
00104, 00110, 00002, 00000;
00104, 00110, 00003, 00000;
00104, 00110, 00004, 00000;
00104, 00110, 00005, 00000;
00104, 00110, 00006, 00000;
00104, 00110, 00007, 00000;
00104, 00110, 00008, 00000;
00104, 00110, 00009, 00000;
00104, 00110, 00010, 00000;
00104, 00110, 00011, 00000;
00104, 00110, 00012, 00000;
00104, 00110, 00013, 00000;
00104, 00110, 00014, 00000;
00104, 00110, 00015, 00000;
00104, 00110, 00016, 00000;
00104, 00110, 00017, 00000;
00104, 00110, 00018, 00000;
00104, 00110, 00019, 00000;
00104, 00110, 00020, 00000;
00104, 00110, 00021, 00000;
00104, 00110, 00022, 00000;
00104, 00110, 00023, 00000;
00104, 00110, 00024, 00000;
00104, 00110, 00025, 00000;
00104, 00110, 00026, 00000;
00104, 00110, 00027, 00000;
00104, 00110, 00028, 00000;
00104, 00110, 00029, 00000;
00104, 00110, 00030, 00000;
00104, 00111, 00001, 00000;
00104, 00111, 00002, 00000;
00104, 00111, 00003, 00000;
00104, 00111, 00004, 00000;
00104, 00111, 00005, 00000;
00104, 00111, 00006, 00000;
00104, 00111, 00007, 00000;
00104, 00111, 00008, 00000;
00104, 00111, 00009, 00000;
00104, 00111, 00010, 00000;
00104, 00111, 00011, 00000;
00104, 00111, 00012, 00000;
00104, 00111, 00013, 00000;
00104, 00111, 00014, 00000;
00104, 00111, 00015, 00000;
00104, 00111, 00016, 00000;
00104, 00111, 00017, 00000;
00104, 00111, 00018, 00000;
00104, 00111, 00019, 00000;
00104, 00111, 00020, 00000;
00104, 00111, 00021, 00000;
00104, 00111, 00022, 00000;
00104, 00111, 00023, 00000;
00104, 00111, 00024, 00000;
00104, 00111, 00025, 00000;
00104, 00111, 00026, 00000;
00104, 00111, 00027, 00000;
00104, 00111, 00028, 00000;
00104, 00111, 00029, 00000;
00104, 00111, 00030, 00000;
00104, 00112, 00001, 00000;
00104, 00112, 00002, 00000;
00104, 00112, 00003, 00000;
00104, 00112, 00004, 00000;
00104, 00112, 00005, 00000;
00104, 00112, 00006, 00000;
00104, 00112, 00007, 00000;
00104, 00112, 00008, 00000;
00104, 00112, 00009, 00000;
00104, 00112, 00010, 00000;
00104, 00112, 00011, 00000;
00104, 00112, 00012, 00000;
00104, 00112, 00013, 00000;
00104, 00112, 00014, 00000;
00104, 00112, 00015, 00000;
00104, 00112, 00016, 00000;
00104, 00112, 00017, 00000;
00104, 00112, 00018, 00000;
00104, 00112, 00019, 00000;
00104, 00112, 00020, 00000;
00104, 00112, 00021, 00000;
00104, 00112, 00022, 00000;
00104, 00112, 00023, 00000;
00104, 00112, 00024, 00000;
00104, 00112, 00025, 00000;
00104, 00112, 00026, 00000;
00104, 00112, 00027, 00000;
00104, 00112, 00028, 00000;
00104, 00112, 00029, 00000;
00104, 00112, 00030, 00000;
00104, 00113, 00001, 00000;
00104, 00113, 00002, 00000;
00104, 00113, 00003, 00000;
00104, 00113, 00004, 00000;
00104, 00113, 00005, 00000;
00104, 00113, 00006, 00000;
00104, 00113, 00007, 00000;
00104, 00113, 00008, 00000;
00104, 00113, 00009, 00000;
00104, 00113, 00010, 00000;
00104, 00113, 00011, 00000;
00104, 00113, 00012, 00000;
00104, 00113, 00013, 00000;
00104, 00113, 00014, 00000;
00104, 00113, 00015, 00000;
00104, 00113, 00016, 00000;
00104, 00113, 00017, 00000;
00104, 00113, 00018, 00000;
00104, 00113, 00019, 00000;
00104, 00113, 00020, 00000;
00104, 00113, 00021, 00000;
00104, 00113, 00022, 00000;
00104, 00113, 00023, 00000;
00104, 00113, 00024, 00000;
00104, 00113, 00025, 00000;
00104, 00113, 00026, 00000;
00104, 00113, 00027, 00000;
00104, 00113, 00028, 00000;
00104, 00113, 00029, 00000;
00104, 00113, 00030, 00000;
; ****************************
; mnTank
;*****************************
;00105, 00000, 00000, 00000;
;****************************
; System Manager
;*****************************
00110, 00003, 00000, 00000;
00110, 00004, 00000, 00000;
00110, 00005, 00000, 00000;
; ****************************
; mnKanLink
;*****************************
00113, 00001, 00000, 00000;
00113, 00002, 00000, 00000;
00113, 00003, 00000, 00000;
00113, 00004, 00000, 00000;
00113, 00101, 00000, 00000;
; ****************************
; fnDrive
;*****************************
00301, 01000, 00000, 00000;
00301, 01001, 00000, 00000;
00301, 01010, 00000, 00000;
00301, 01011, 00000, 00000;
00301, 01020, 00000, 00000;
00301, 01021, 00000, 00000;
00301, 01030, 00000, 00000;
; ****************************
; fnWater
;*****************************
00302, 01041, 00001, 00000;
00302, 01041, 00002, 00000;
00302, 01041, 00003, 00000;
00302, 01041, 00004, 00000;
00302, 01041, 00005, 00000;
00302, 01041, 00006, 00000;
00302, 01041, 00007, 00000;
00302, 01041, 00008, 00000;
00302, 01041, 00009, 00000;
00302, 01041, 00010, 00000;
00302, 01041, 00011, 00000;
00302, 01041, 00012, 00000;
00302, 01041, 00013, 00000;
00302, 01041, 00014, 00000;
00302, 01041, 00015, 00000;
00302, 01041, 00016, 00000;
00302, 01041, 00017, 00000;
00302, 01041, 00018, 00000;
00302, 01041, 00019, 00000;
00302, 01041, 00020, 00000;
00302, 01041, 00021, 00000;
00302, 01041, 00022, 00000;
00302, 01041, 00023, 00000;
00302, 01041, 00024, 00000;
00302, 01041, 00025, 00000;
00302, 01041, 00026, 00000;
00302, 01041, 00027, 00000;
00302, 01041, 00028, 00000;
00302, 01041, 00029, 00000;
00302, 01041, 00030, 00000;
00302, 01041, 00031, 00000;
00302, 01041, 00032, 00000;
00302, 01041, 00033, 00000;
00302, 01041, 00034, 00000;
00302, 01041, 00035, 00000;
00302, 01041, 00036, 00000;
00302, 01041, 00037, 00000;
00302, 01041, 00038, 00000;
00302, 01041, 00039, 00000;
00302, 01041, 00040, 00000;
00302, 01041, 00041, 00000;
00302, 01041, 00042, 00000;
00302, 01041, 00043, 00000;
00302, 01041, 00044, 00000;
00302, 01041, 00045, 00000;
00302, 01041, 00046, 00000;
00302, 01041, 00047, 00000;
00302, 01041, 00048, 00000;
00302, 01041, 00049, 00000;
00302, 01041, 00050, 00000;
00302, 01041, 00051, 00000;
00302, 01041, 00052, 00000;
00302, 01041, 00053, 00000;
00302, 01041, 00054, 00000;
00302, 01041, 00055, 00000;
00302, 01041, 00056, 00000;
00302, 01041, 00057, 00000;
00302, 01041, 00058, 00000;
00302, 01041, 00059, 00000;
00302, 01041, 00060, 00000;
00302, 01042, 00001, 00000;
00302, 01042, 00002, 00000;
00302, 01042, 00003, 00000;
00302, 01042, 00004, 00000;
00302, 01042, 00005, 00000;
00302, 01042, 00006, 00000;
00302, 01042, 00007, 00000;
00302, 01042, 00008, 00000;
00302, 01042, 00009, 00000;
00302, 01042, 00010, 00000;
00302, 01042, 00011, 00000;
00302, 01042, 00012, 00000;
00302, 01042, 00013, 00000;
00302, 01042, 00014, 00000;
00302, 01042, 00015, 00000;
00302, 01042, 00016, 00000;
00302, 01042, 00017, 00000;
00302, 01042, 00018, 00000;
00302, 01042, 00019, 00000;
00302, 01042, 00020, 00000;
00302, 01042, 00021, 00000;
00302, 01042, 00022, 00000;
00302, 01042, 00023, 00000;
00302, 01042, 00024, 00000;
00302, 01042, 00025, 00000;
00302, 01042, 00026, 00000;
00302, 01042, 00027, 00000;
00302, 01042, 00028, 00000;
00302, 01042, 00029, 00000;
00302, 01042, 00030, 00000;
00302, 01042, 00031, 00000;
00302, 01042, 00032, 00000;
00302, 01042, 00033, 00000;
00302, 01042, 00034, 00000;
00302, 01042, 00035, 00000;
00302, 01042, 00036, 00000;
00302, 01042, 00037, 00000;
00302, 01042, 00038, 00000;
00302, 01042, 00039, 00000;
00302, 01042, 00040, 00000;
00302, 01042, 00041, 00000;
00302, 01042, 00042, 00000;
00302, 01042, 00043, 00000;
00302, 01042, 00044, 00000;
00302, 01042, 00045, 00000;
00302, 01042, 00046, 00000;
00302, 01042, 00047, 00000;
00302, 01042, 00048, 00000;
00302, 01042, 00049, 00000;
00302, 01042, 00050, 00000;
00302, 01042, 00051, 00000;
00302, 01042, 00052, 00000;
00302, 01042, 00053, 00000;
00302, 01042, 00054, 00000;
00302, 01042, 00055, 00000;
00302, 01042, 00056, 00000;
00302, 01042, 00057, 00000;
00302, 01042, 00058, 00000;
00302, 01042, 00059, 00000;
00302, 01042, 00060, 00000;
00302, 06666, 00001, 00000;
00302, 06666, 00002, 00000;
00302, 06666, 00003, 00000;
00302, 06666, 00004, 00000;
00302, 06666, 00005, 00000;
00302, 06666, 00006, 00000;
00302, 06666, 00007, 00000;
00302, 06666, 00008, 00000;
00302, 06666, 00009, 00000;
00302, 06666, 00010, 00000;
00302, 06666, 00011, 00000;
00302, 06666, 00012, 00000;
00302, 06666, 00013, 00000;
00302, 06666, 00014, 00000;
00302, 06666, 00015, 00000;
00302, 06666, 00016, 00000;
00302, 06666, 00017, 00000;
00302, 06666, 00018, 00000;
00302, 06666, 00019, 00000;
00302, 06666, 00020, 00000;
00302, 06666, 00021, 00000;
00302, 06666, 00022, 00000;
00302, 06666, 00023, 00000;
00302, 06666, 00024, 00000;
00302, 06666, 00025, 00000;
00302, 06666, 00026, 00000;
00302, 06666, 00027, 00000;
00302, 06666, 00028, 00000;
00302, 06666, 00029, 00000;
00302, 06666, 00030, 00000;
00302, 06666, 00031, 00000;
00302, 06666, 00032, 00000;
00302, 06666, 00033, 00000;
00302, 06666, 00034, 00000;
00302, 06666, 00035, 00000;
00302, 06666, 00036, 00000;
00302, 06666, 00037, 00000;
00302, 06666, 00038, 00000;
00302, 06666, 00039, 00000;
00302, 06666, 00040, 00000;
00302, 06666, 00041, 00000;
00302, 06666, 00042, 00000;
00302, 06666, 00043, 00000;
00302, 06666, 00044, 00000;
00302, 06666, 00045, 00000;
00302, 06666, 00046, 00000;
00302, 06666, 00047, 00000;
00302, 06666, 00048, 00000;
00302, 06666, 00049, 00000;
00302, 06666, 00050, 00000;
00302, 06666, 00051, 00000;
00302, 06666, 00052, 00000;
00302, 06666, 00053, 00000;
00302, 06666, 00054, 00000;
00302, 06666, 00055, 00000;
00302, 06666, 00056, 00000;
00302, 06666, 00057, 00000;
00302, 06666, 00058, 00000;
00302, 06666, 00059, 00000;
00302, 06666, 00060, 00000;
; ****************************
; fnHeater
;*****************************
00303, 01032, 00001, 00000;
00303, 01032, 00002, 00000;
00303, 01032, 00003, 00000;
00303, 01032, 00004, 00000;
00303, 01032, 00005, 00000;
00303, 01032, 00006, 00000;
00303, 01032, 00007, 00000;
00303, 01032, 00008, 00000;
00303, 01032, 00009, 00000;
00303, 01033, 00001, 00000;
00303, 01033, 00002, 00000;
00303, 01033, 00003, 00000;
00303, 01033, 00004, 00000;
00303, 01033, 00005, 00000;
00303, 01033, 00006, 00000;
00303, 01033, 00007, 00000;
00303, 01033, 00008, 00000;
00303, 01033, 00009, 00000;
00303, 06666, 00001, 00000;
00303, 06666, 00002, 00000;
00303, 06666, 00003, 00000;
00303, 06666, 00004, 00000;
00303, 06666, 00005, 00000;
00303, 06666, 00006, 00000;
00303, 06666, 00007, 00000;
00303, 06666, 00008, 00000;
00303, 06666, 00009, 00000;
; ****************************
; fnDos
;*****************************
00304, 01001, 00000, 00000;
; ****************************
; svDrive
;*****************************
00501, 01003, 00000, 00000;
00501, 01005, 00000, 00000;
00501, 01009, 00000, 00000;
00501, 01011, 00000, 00000;
00501, 01020, 00000, 00000;
00501, 01021, 00000, 00000;
00501, 01022, 00000, 00000;
00501, 01023, 00000, 00000;
00501, 01024, 00000, 00000;
00501, 01025, 00000, 00000;
00501, 01026, 00000, 00000;
00501, 01027, 00000, 00000;
00501, 01028, 00000, 00000;
00501, 01030, 00000, 00000;
; ****************************
; svRoute
;*****************************
00502, 01017, 00001, 00000;
00502, 01017, 00002, 00000;
00502, 01017, 00003, 00000;
00502, 01017, 00004, 00000;
00502, 01017, 00005, 00000;
00502, 01017, 00006, 00000;
00502, 01017, 00007, 00000;
00502, 01017, 00008, 00000;
00502, 01017, 00009, 00000;
00502, 01017, 00010, 00000;
00502, 01017, 00011, 00000;
00502, 01017, 00012, 00000;
00502, 01017, 00013, 00000;
00502, 01017, 00014, 00000;
00502, 01017, 00015, 00000;
00502, 01017, 00016, 00000;
00502, 01017, 00017, 00000;
00502, 01017, 00018, 00000;
00502, 01017, 00019, 00000;
00502, 01017, 00020, 00000;
00502, 01017, 00021, 00000;
00502, 01017, 00022, 00000;
00502, 01017, 00023, 00000;
00502, 01017, 00024, 00000;
00502, 01017, 00025, 00000;
00502, 01017, 00026, 00000;
00502, 01017, 00027, 00000;
00502, 01017, 00028, 00000;
00502, 01017, 00029, 00000;
00502, 01017, 00030, 00000;
00502, 01017, 00031, 00000;
00502, 01017, 00032, 00000;
00502, 01017, 00033, 00000;
00502, 01017, 00034, 00000;
00502, 01017, 00035, 00000;
00502, 01017, 00036, 00000;
00502, 01017, 00037, 00000;
00502, 01017, 00038, 00000;
00502, 01017, 00039, 00000;
00502, 01017, 00040, 00000;
00502, 01017, 00041, 00000;
00502, 01017, 00042, 00000;
00502, 01017, 00043, 00000;
00502, 01017, 00044, 00000;
00502, 01017, 00045, 00000;
00502, 01017, 00046, 00000;
00502, 01017, 00047, 00000;
00502, 01017, 00048, 00000;
00502, 01017, 00049, 00000;
00502, 01017, 00050, 00000;
00502, 01017, 00051, 00000;
00502, 01017, 00052, 00000;
00502, 01017, 00053, 00000;
00502, 01017, 00054, 00000;
00502, 01017, 00055, 00000;
00502, 01017, 00056, 00000;
00502, 01017, 00057, 00000;
00502, 01017, 00058, 00000;
00502, 01017, 00059, 00000;
00502, 01017, 00060, 00000;
00502, 01017, 00061, 00000;
00502, 01017, 00062, 00000;
00502, 01017, 00063, 00000;
00502, 01017, 00064, 00000;
00502, 01017, 00065, 00000;
00502, 01017, 00066, 00000;
00502, 01017, 00067, 00000;
00502, 01017, 00068, 00000;
00502, 01017, 00069, 00000;
00502, 01017, 00070, 00000;
00502, 01018, 00001, 00000;
00502, 01018, 00002, 00000;
00502, 01018, 00003, 00000;
00502, 01018, 00004, 00000;
00502, 01018, 00005, 00000;
00502, 01018, 00006, 00000;
00502, 01018, 00007, 00000;
00502, 01018, 00008, 00000;
00502, 01018, 00009, 00000;
00502, 01018, 00010, 00000;
00502, 01018, 00011, 00000;
00502, 01018, 00012, 00000;
00502, 01018, 00013, 00000;
00502, 01018, 00014, 00000;
00502, 01018, 00015, 00000;
00502, 01018, 00016, 00000;
00502, 01018, 00017, 00000;
00502, 01018, 00018, 00000;
00502, 01018, 00019, 00000;
00502, 01018, 00020, 00000;
00502, 01018, 00021, 00000;
00502, 01018, 00022, 00000;
00502, 01018, 00023, 00000;
00502, 01018, 00024, 00000;
00502, 01018, 00025, 00000;
00502, 01018, 00026, 00000;
00502, 01018, 00027, 00000;
00502, 01018, 00028, 00000;
00502, 01018, 00029, 00000;
00502, 01018, 00030, 00000;
00502, 01018, 00031, 00000;
00502, 01018, 00032, 00000;
00502, 01018, 00033, 00000;
00502, 01018, 00034, 00000;
00502, 01018, 00035, 00000;
00502, 01018, 00036, 00000;
00502, 01018, 00037, 00000;
00502, 01018, 00038, 00000;
00502, 01018, 00039, 00000;
00502, 01018, 00040, 00000;
00502, 01018, 00041, 00000;
00502, 01018, 00042, 00000;
00502, 01018, 00043, 00000;
00502, 01018, 00044, 00000;
00502, 01018, 00045, 00000;
00502, 01018, 00046, 00000;
00502, 01018, 00047, 00000;
00502, 01018, 00048, 00000;
00502, 01018, 00049, 00000;
00502, 01018, 00050, 00000;
00502, 01018, 00051, 00000;
00502, 01018, 00052, 00000;
00502, 01018, 00053, 00000;
00502, 01018, 00054, 00000;
00502, 01018, 00055, 00000;
00502, 01018, 00056, 00000;
00502, 01018, 00057, 00000;
00502, 01018, 00058, 00000;
00502, 01018, 00059, 00000;
00502, 01018, 00060, 00000;
00502, 01018, 00061, 00000;
00502, 01018, 00062, 00000;
00502, 01018, 00063, 00000;
00502, 01018, 00064, 00000;
00502, 01018, 00065, 00000;
00502, 01018, 00066, 00000;
00502, 01018, 00067, 00000;
00502, 01018, 00068, 00000;
00502, 01018, 00069, 00000;
00502, 01018, 00070, 00000;
00502, 06666, 00001, 00000;
00502, 06666, 00002, 00000;
00502, 06666, 00003, 00000;
00502, 06666, 00004, 00000;
00502, 06666, 00005, 00000;
00502, 06666, 00006, 00000;
00502, 06666, 00007, 00000;
00502, 06666, 00008, 00000;
00502, 06666, 00009, 00000;
00502, 06666, 00010, 00000;
00502, 06666, 00011, 00000;
00502, 06666, 00012, 00000;
00502, 06666, 00013, 00000;
00502, 06666, 00014, 00000;
00502, 06666, 00015, 00000;
00502, 06666, 00016, 00000;
00502, 06666, 00017, 00000;
00502, 06666, 00018, 00000;
00502, 06666, 00019, 00000;
00502, 06666, 00020, 00000;
00502, 06666, 00021, 00000;
00502, 06666, 00022, 00000;
00502, 06666, 00023, 00000;
00502, 06666, 00024, 00000;
00502, 06666, 00025, 00000;
00502, 06666, 00026, 00000;
00502, 06666, 00027, 00000;
00502, 06666, 00028, 00000;
00502, 06666, 00029, 00000;
00502, 06666, 00030, 00000;
00502, 06666, 00031, 00000;
00502, 06666, 00032, 00000;
00502, 06666, 00033, 00000;
00502, 06666, 00034, 00000;
00502, 06666, 00035, 00000;
00502, 06666, 00036, 00000;
00502, 06666, 00037, 00000;
00502, 06666, 00038, 00000;
00502, 06666, 00039, 00000;
00502, 06666, 00040, 00000;
00502, 06666, 00041, 00000;
00502, 06666, 00042, 00000;
00502, 06666, 00043, 00000;
00502, 06666, 00044, 00000;
00502, 06666, 00045, 00000;
00502, 06666, 00046, 00000;
00502, 06666, 00047, 00000;
00502, 06666, 00048, 00000;
00502, 06666, 00049, 00000;
00502, 06666, 00050, 00000;
00502, 06666, 00051, 00000;
00502, 06666, 00052, 00000;
00502, 06666, 00053, 00000;
00502, 06666, 00054, 00000;
00502, 06666, 00055, 00000;
00502, 06666, 00056, 00000;
00502, 06666, 00057, 00000;
00502, 06666, 00058, 00000;
00502, 06666, 00059, 00000;
00502, 06666, 00060, 00000;
00502, 06666, 00061, 00000;
00502, 06666, 00062, 00000;
00502, 06666, 00063, 00000;
00502, 06666, 00064, 00000;
00502, 06666, 00065, 00000;
00502, 06666, 00066, 00000;
00502, 06666, 00067, 00000;
00502, 06666, 00068, 00000;
00502, 06666, 00069, 00000;
00502, 06666, 00070, 00000;
; ****************************
; svWetAcc
;*****************************
00503, 06666, 00001, 00000;
00503, 06666, 00002, 00000;
00503, 06666, 00003, 00000;
00503, 06666, 00004, 00000;
00503, 06666, 00005, 00000;
00503, 06666, 00006, 00000;
00503, 06666, 00007, 00000;
00503, 06666, 00008, 00000;
00503, 06666, 00009, 00000;
00503, 06666, 00010, 00000;
00503, 06666, 00011, 00000;
00503, 06666, 00012, 00000;
00503, 06666, 00013, 00000;
00503, 06666, 00014, 00000;
00503, 06666, 00015, 00000;
00503, 06666, 00016, 00000;
00503, 06666, 00017, 00000;
00503, 06666, 00018, 00000;
00503, 06666, 00019, 00000;
00503, 06666, 00020, 00000;
00503, 06666, 00021, 00000;
00503, 06666, 00022, 00000;
00503, 06666, 00023, 00000;
00503, 06666, 00024, 00000;
00503, 06666, 00025, 00000;
00503, 06666, 00026, 00000;
00503, 06666, 00027, 00000;
00503, 06666, 00028, 00000;
00503, 06666, 00029, 00000;
00503, 06666, 00030, 00000;
00503, 06666, 00031, 00000;
00503, 06666, 00032, 00000;
00503, 06666, 00033, 00000;
00503, 06666, 00034, 00000;
00503, 06666, 00035, 00000;
00503, 06666, 00036, 00000;
00503, 06666, 00037, 00000;
00503, 06666, 00038, 00000;
00503, 06666, 00039, 00000;
00503, 06666, 00040, 00000;
00503, 06666, 00041, 00000;
00503, 06666, 00042, 00000;
00503, 06666, 00043, 00000;
00503, 06666, 00044, 00000;
00503, 06666, 00045, 00000;
00503, 06666, 00046, 00000;
00503, 06666, 00047, 00000;
00503, 06666, 00048, 00000;
00503, 06666, 00049, 00000;
00503, 06666, 00050, 00000;
00503, 06666, 00051, 00000;
00503, 06666, 00052, 00000;
00503, 06666, 00053, 00000;
00503, 06666, 00054, 00000;
00503, 06666, 00055, 00000;
00503, 06666, 00056, 00000;
00503, 06666, 00057, 00000;
00503, 06666, 00058, 00000;
00503, 06666, 00059, 00000;
00503, 06666, 00060, 00000;
00503, 06666, 00061, 00000;
00503, 06666, 00062, 00000;
00503, 06666, 00063, 00000;
00503, 06666, 00064, 00000;
00503, 06666, 00065, 00000;
00503, 06666, 00066, 00000;
00503, 06666, 00067, 00000;
00503, 06666, 00068, 00000;
00503, 06666, 00069, 00000;
00503, 06666, 00070, 00000;
; ****************************
; hlEncoder
;*****************************
00701, 00201, 00000, 00000;
; ****************************
; hlDSwIn
;*****************************
; Hat keine Fehlermeldungen.
; ****************************
; hlFC
;*****************************
00703, 00201, 00000, 00000;
00703, 00202, 00000, 00000;
00703, 01002, 00000, 00000;
00703, 01003, 00000, 00000;
; ****************************
; hlValve
;*****************************
; Es gibt keine Fehler
; ****************************
; hlMotor
;*****************************
00705, 01004, 00001, 00000;
00705, 01004, 00002, 00000;
00705, 01004, 00003, 00000;
00705, 01004, 00004, 00000;
00705, 01004, 00005, 00000;
00705, 01004, 00006, 00000;
00705, 01004, 00007, 00000;
00705, 01004, 00008, 00000;
00705, 01004, 00009, 00000;
00705, 01004, 00010, 00000;
00705, 01004, 00011, 00000;
00705, 01004, 00012, 00000;
00705, 01004, 00013, 00000;
00705, 01004, 00014, 00000;
00705, 01004, 00015, 00000;
00705, 01004, 00016, 00000;
00705, 01004, 00017, 00000;
00705, 01004, 00018, 00000;
00705, 01004, 00019, 00000;
00705, 01004, 00020, 00000;
00705, 01005, 00001, 00000;
00705, 01005, 00002, 00000;
00705, 01005, 00003, 00000;
00705, 01005, 00004, 00000;
00705, 01005, 00005, 00000;
00705, 01005, 00006, 00000;
00705, 01005, 00007, 00000;
00705, 01005, 00008, 00000;
00705, 01005, 00009, 00000;
00705, 01005, 00010, 00000;
00705, 01005, 00011, 00000;
00705, 01005, 00012, 00000;
00705, 01005, 00013, 00000;
00705, 01005, 00014, 00000;
00705, 01005, 00015, 00000;
00705, 01005, 00016, 00000;
00705, 01005, 00017, 00000;
00705, 01005, 00018, 00000;
00705, 01005, 00019, 00000;
00705, 01005, 00020, 00000;
; ****************************
; hlRate
;*****************************
; Es gibt keine Fehler
; ****************************
; hlNiveau
;*****************************
00708, 01001, 00001, 00000;
00708, 01001, 00002, 00000;
00708, 01001, 00003, 00000;
00708, 01001, 00004, 00000;
00708, 01001, 00005, 00000;
00708, 01001, 00006, 00000;
00708, 01001, 00007, 00000;
00708, 01001, 00008, 00000;
00708, 01001, 00009, 00000;
00708, 01001, 00010, 00000;
00708, 01001, 00011, 00000;
00708, 01001, 00012, 00000;
00708, 01001, 00013, 00000;
00708, 01001, 00014, 00000;
00708, 01002, 00001, 00000;
00708, 01002, 00002, 00000;
00708, 01002, 00003, 00000;
00708, 01002, 00004, 00000;
00708, 01002, 00005, 00000;
00708, 01002, 00006, 00000;
00708, 01002, 00007, 00000;
00708, 01002, 00008, 00000;
00708, 01002, 00009, 00000;
00708, 01002, 00010, 00000;
00708, 01002, 00011, 00000;
00708, 01002, 00012, 00000;
00708, 01002, 00013, 00000;
00708, 01002, 00014, 00000;
; ****************************
; hlTemp
;*****************************
00709, 01001, 00001, 00000;
00709, 01001, 00002, 00000;
00709, 01001, 00003, 00000;
00709, 01001, 00004, 00000;
00709, 01001, 00005, 00000;
00709, 01001, 00006, 00000;
00709, 01001, 00007, 00000;
00709, 01001, 00008, 00000;
00709, 01001, 00009, 00000;
00709, 01001, 00010, 00000;
00709, 01001, 00011, 00000;
00709, 01001, 00012, 00000;
00709, 01001, 00013, 00000;
00709, 01001, 00014, 00000;
00709, 01001, 00015, 00000;
00709, 01002, 00001, 00000;
00709, 01002, 00002, 00000;
00709, 01002, 00003, 00000;
00709, 01002, 00004, 00000;
00709, 01002, 00005, 00000;
00709, 01002, 00006, 00000;
00709, 01002, 00007, 00000;
00709, 01002, 00008, 00000;
00709, 01002, 00009, 00000;
00709, 01002, 00010, 00000;
00709, 01002, 00011, 00000;
00709, 01002, 00012, 00000;
00709, 01002, 00013, 00000;
00709, 01002, 00014, 00000;
00709, 01002, 00015, 00000;
00709, 01006, 00001, 00000;
00709, 01006, 00002, 00000;
00709, 01006, 00003, 00000;
00709, 01006, 00004, 00000;
00709, 01006, 00005, 00000;
00709, 01006, 00006, 00000;
00709, 01006, 00007, 00000;
00709, 01006, 00008, 00000;
00709, 01006, 00009, 00000;
00709, 01006, 00010, 00000;
00709, 01006, 00011, 00000;
00709, 01006, 00012, 00000;
00709, 01006, 00013, 00000;
00709, 01006, 00014, 00000;
00709, 01006, 00015, 00000;
; ****************************
; hlDos
;*****************************
00711, 01001, 00000, 00000;
00711, 01002, 00000, 00000;
00711, 01003, 00000, 00000;
00711, 01004, 00000, 00000;
00711, 01005, 00000, 00000;
00711, 01006, 00000, 00000;
00711, 01007, 00000, 00000;
; ****************************
; hlHWCont
;*****************************
00713, 00001, 00000, 00000;
00713, 00010, 00000, 00000;
00713, 00012, 00000, 00000;
00713, 00101, 00000, 00000;
00713, 00111, 00000, 00000;
; ****************************
; hlGrease
;*****************************
00714, 00001, 00000, 00000;
00714, 00011, 00000, 00000;
00714, 00021, 00000, 00000;
00714, 08888, 00000, 00000;
; ****************************
; hlSafety
;*****************************
00717, 00100, 00001, 00000;
00717, 00100, 00002, 00000;
00717, 00101, 00001, 00000;
00717, 00101, 00002, 00000;
00717, 00102, 00001, 00000;
00717, 00102, 00002, 00000;
00717, 00103, 00001, 00000;
00717, 00103, 00002, 00000;
```

### Package Logical/Mewa/KGFrameworkShare/Pkg_hlKanLinkUser - Kanlink User

### Library Logical/Mewa/KGFrameworkShare/Pkg_hlKanLinkUser/KL_UserLib (IEC, version 0.91.0) - Kanlink User Library

#### KL_UserLib.var - Exported constants
```iecst
(********************************************************************
 * COPYRIGHT -- Herbert Kannegiesser GmbH
 ********************************************************************
 * Library: WL_UserLib
 * File: WL_UserLib.var
 * Author: stahlhut
 * Created: January 10, 2012
 ********************************************************************
 * Constants of library WL_UserLib
 ********************************************************************)
VAR CONSTANT
	HLKANLINK_MAX_CLIENTCONNS : UINT := 10; (*Anzahl der Clienten *)
	HLKANLINK_MAX_SERVERCONNS : UINT := 10; (*Anzahl der Server *)
END_VAR
```


- Library Logical/Mewa/KGFrameworkShare/Pkg_mnTestUser/libTestUse (IEC) - Userlibrary für Testadapter (no source held here)

- Program Logical/Mewa/KGFrameworkShare/Pkg_mnTestUser/mnTestUser (IEC) - Initialisierung des Test (no source held here)

Listed in the project but not available here: Logical/Reference/4_ppn1/ppn.var, Logical/Reference/6_pwb1, Logical/Reference/7_pwb2, Logical/Reference/10_pup2, Logical/Reference/11_pup3, Logical/Reference/14_pup6, Logical/Reference/19_pp5, Logical/Reference/20_pp6/pp.var, Logical/Reference/21_pp7, Logical/Reference/24_pp10, Logical/Reference/25_pp11, Logical/Reference/29_pp17, Logical/Reference/34_picd5, Logical/Reference/36_picu7, Logical/Reference/38_picu9, Logical/Reference/39_picu10, Logical/Reference/41_picd12/picu.var, Logical/Reference/42_picd13, Logical/Sequences/10ms/zzPrimSearch/zzPrimSearch.typ, Logical/Sequences/10ms/zzStatus/zzstatus.ab, Logical/Sequences/10ms/1_stnsa/1_stnsaInit.ab, Logical/Sequences/10ms/1_stnsa/1_stnsa.var, Logical/Sequences/10ms/2_belt1/2_belt1.var, Logical/Sequences/10ms/4_spn1/4_spn1Init.ab, Logical/Sequences/10ms/4_spn1/4_spn1.var, Logical/Sequences/10ms/5_spf1/5_spf1Init.ab, Logical/Sequences/10ms/5_spf1/5_spf1.var, Logical/Sequences/10ms/6_sdc1/6_sdc1Init.ab, Logical/Sequences/10ms/9_sic1/9_spc1Init.ab, Logical/Sequences/10ms/11_bsoff/11_bsoffInit.ab, Logical/Sequences/10ms/zzForceO/zzforceo.var, Logical/Sequences/10ms/zzForceO/zzforceo.ab, Logical/Sequences/10ms/zzOk/zzok.var, Logical/Sequences/10ms/zzOk/zzok.ab, Logical/Sequences/200ms/zzClearMem/zzclrmem.var, Logical/Sequences/200ms/zzClearMem/zzclrmem.ab, Logical/Sequences/200ms/zzWeigh/zzweigh.typ, Logical/Sequences/200ms/zzStn_Q/zzstn_q.var, Logical/Sequences/200ms/zzTime/zztime.var, Logical/Sequences/200ms/zzTime/zztime.ab, Logical/Sequences/zzstnmix/zzstnmix.var, Logical/Sequences/zzstnmix/zzstnmixInit.ab, Logical/Sequences/zzstnmix/zzstnmixCyclic.ab, Logical/Sequences/zzstatus/zzstatusInit.ab, Logical/Sequences/zzstatus/zzstatusCyclic.ab, Logical/Sequences/zzstnser/zzstnserInit.ab, Logical/Sequences/zztc2str/zztc2str.var, Logical/Sequences/zztc2str/zztc2strInit.ab, Logical/Sequences/zztc2str/zztc2strCyclic.ab, Logical/Sequences/zzforcei/zzforcei.var, Logical/Sequences/zzforcei/zzforceiInit.ab, Logical/Sequences/zzforcei/zzforceiCyclic.ab, Logical/Sequences/zzbagsfl/zzbagsfl.var, Logical/Sequences/zzbagsfl/zzbagsflInit.ab, Logical/Sequences/zzbitcal/zzbitcalCyclic.ab, Logical/Sequences/zcusfifo/zcusfifo.var, Logical/Sequences/zcusfifo/zcusfifoInit.ab, Logical/Sequences/zzindi, Logical/Sequences/zzforceo/zzforceo.var, Logical/Sequences/zzforceo/zzforceoCyclic.ab, Logical/Sequences/zztc2end, Logical/Sequences/zzio, Logical/Sequences/zzuld_3/zzuld_3.var, Logical/Sequences/zzuld_3/zzuld_3Init.ab, Logical/Sequences/zzstn_q/zzstn_q.var, Logical/Sequences/zzstn_q/zzstn_qInit.ab, Logical/Sequences/can_live/can_liveInit.ab, Logical/Libraries/IecCheck/IecCheck.fun, Logical/a_flx_io, Logical/Timestamp/zzGetTime/zzGetTime.typ, Logical/Timestamp/zzGetTime/zzGetTime.var, Logical/Data_BackUp/DataBackUp/DataBackUp.typ, Logical/Data_BackUp/DataBackUp/DataBackUp.var, Logical/Data_BackUp/DataBackUp/DataBackUp.fun, Logical/SQL/zzSQLDriver/zzSQLDriver.ab, Logical/SQL/zzSQLDriver/zzSQLDriver.var, Logical/zztc2end/zztc2endCyclic.ab, Logical/zztc2end/zztc2endInit.ab, Logical/zztc2end/zztc2end.var, Logical/zzreport/zzreportCyclic.ab, Logical/zzreport/zzreportInit.ab, Logical/zzreport/zzreport.var, Logical/zztime/zztimeCyclic.ab, Logical/zztime/zztime.var, Logical/Mewa/200ms/CAN/can.var, Logical/Mewa/200ms/CAN/can_stn/can_stn.var, Logical/Mewa/200ms/CAN/can_live/can_live.var, Logical/Mewa/KGFramework/Pkg_KGStandard/KG_Cmd.typ, Logical/Mewa/KGFramework/Pkg_KGStandard/KG_Cmd.var, Logical/Mewa/KGFramework/Pkg_KGStandard/Stat.typ, Logical/Mewa/KGFramework/Pkg_KGStandard/Stat.var, Logical/Mewa/KGFramework/Pkg_KGStandard/utfNames.typ, Logical/Mewa/KGFramework/Pkg_KGStandard/kgbom.var, Logical/Mewa/KGFramework/Pkg_KGStandard/kgMachineState.typ, Logical/Mewa/KGFramework/Pkg_KGStandard/KGstdLib/KGstdLib.typ, Logical/Mewa/KGFramework/Pkg_KGStandard/KGstdLib/kgMachinetyp.typ, Logical/Mewa/KGFramework/Pkg_KGStandard/KGstdLib/kgitoa_udint.st, Logical/Mewa/KGFramework/Pkg_KGStandard/KGstdLib/kgatoi_udint.st, Logical/Mewa/KGFramework/Pkg_KGStandard/KGstdLib/kgatoi_uint.st, Logical/Mewa/KGFramework/Pkg_KGStandard/KGstdLib/kgInitBatchNoLong.st, Logical/Mewa/KGFramework/Pkg_KGStandard/KGstdLib/kgNextBatchNoLong.st, Logical/Mewa/KGFramework/Pkg_KGStandard/KGstdLib/kgGetMacAdress.st, Logical/Mewa/KGFramework/Pkg_KGStandard/KGstdLib/kgGetBatchNoUnique.st, Logical/Mewa/KGFramework/Pkg_KGStandard/KGstdLib/kgBatchNoToUDINT.st, Logical/Mewa/KGFramework/Pkg_KGStandard/KGstdLib/kgUSINT16toGUID.st, Logical/Mewa/KGFramework/Pkg_KGStandard/KGstdLib/kgGUIDtoSTRING.st, Logical/Mewa/KGFramework/Pkg_KGStandard/KGstdLib/kgLogLine.st, Logical/Mewa/KGFramework/Pkg_KGStandard/KGstdLib/kgArLogWrite.st, Logical/Mewa/KGFramework/Pkg_KGStandard/KGstdLib/kgRBcreate.st, Logical/Mewa/KGFramework/Pkg_KGStandard/KGstdLib/kgRBinsert.st, Logical/Mewa/KGFramework/Pkg_KGStandard/KGstdLib/kgRBread.st, Logical/Mewa/KGFramework/Pkg_KGStandard/KGstdLib/kgRBloc.st, Logical/Mewa/KGFramework/Pkg_KGStandard/KGstdLib/kgGUIDisZero.st, Logical/Mewa/KGFramework/Pkg_KGStandard/KGstdLib/kgRBbulkloc.st, Logical/Mewa/KGFramework/Pkg_KGStandard/KGstdLib/kgGetLineNumberW3.st, Logical/Mewa/KGFramework/Pkg_KGStandard/KGstdLib/kgGetMachineAdressW3.st, Logical/Mewa/KGFramework/Pkg_KGStandard/KGstdLib/kgCheckDo.st, Logical/Mewa/KGFramework/Pkg_KGStandard/KGstdLib/kgXOR.st, Logical/Mewa/KGFramework/Pkg_mnEth/Pkg_mnEth.var, Logical/Mewa/KGFramework/Pkg_mnCnt/mnCnt/mnCntCyclic.st, Logical/Mewa/KGFramework/Pkg_mnCnt/mnCnt/mnCntInit.st, Logical/Mewa/KGFramework/Pkg_mnCnt/mnCnt/mnCnt.typ, Logical/Mewa/KGFramework/Pkg_mnCnt/mnCnt/mnCnt.var, Logical/Mewa/KGFramework/Pkg_mnMsg/Pkg_mnMsg.typ, Logical/Mewa/KGFramework/Pkg_mnMsg/Pkg_mnMsg.var, Logical/Mewa/KGFramework/Pkg_mnMsg/mnMsg/mnMsgInit.st, Logical/Mewa/KGFramework/Pkg_mnMsg/mnMsg/mnMsg.typ, Logical/Mewa/KGFramework/Pkg_mnMsg/mnMsg/mnMsg.var, Logical/Mewa/KGFramework/Pkg_mnMsg/mnMsg/_actGetOneTurnRB.st, Logical/Mewa/KGFramework/Pkg_mnMsg/mnMsg/_actSetMsgOrMaint.st, Logical/Mewa/KGFramework/Pkg_mnMsg/mnMsg/_actInsertRB.st, Logical/Mewa/KGFramework/Pkg_mnMsg/mnMsg/_actInsertMsgL.st, Logical/Mewa/KGFramework/Pkg_mnMsg/mnMsg/_actStatisticTextLCID.st, Logical/Mewa/KGFramework/Pkg_mnMsg/mnMsg/_actLocMOD.st, Logical/Mewa/KGFramework/Pkg_mnMsg/mnMsg/_actEventClassSel.st, Logical/Mewa/KGFramework/Pkg_mnMsg/KGlibMsg/KGlibMsg.typ, Logical/Mewa/KGFramework/Pkg_mnMsg/KGlibMsg/KGlibMsg.var, Logical/Mewa/KGFramework/Pkg_mnMsg/KGlibMsg/KGlibMsg.fun, Logical/Mewa/KGFramework/Pkg_mnMsg/KGlibMsg/msgBinSearchCfgList.st, Logical/Mewa/KGFramework/Pkg_mnMsg/KGlibMsg/msgInsertMsgLine.st, Logical/Mewa/KGFramework/Pkg_mnMsg/KGlibMsg/msgBinSearchTxtLine.st, Logical/Mewa/KGFramework/Pkg_mnMsg/KGlibMsg/msgBinSearchHelpTxtLine.st, Logical/Mewa/KGFramework/Pkg_mnMsg/KGlibMsg/msgReplSubStr.st, Logical/Mewa/KGFramework/Pkg_mnMsg/KGlibMsg/msgNextChrPos.st, Logical/Mewa/KGFramework/Pkg_mnParam/mnParam/mnParamExit.st, Logical/Mewa/KGFramework/Pkg_mnParam/mnParam/_DefActContainer.st, Logical/Mewa/KGFramework/Pkg_mnParam/mnParam/_BinSearchTxtLine.st, Logical/Mewa/KGFramework/Pkg_mnParam/mnParam/_BinSearchHlpTxtLine.st, Logical/Mewa/KGFramework/Pkg_mnParam/mnParam/_actInterfacePC.st, Logical/Mewa/KGFramework/Pkg_mnParam/mnParam/_actFillNamelist.st, Logical/Mewa/KGFramework/Pkg_mnParam/mnParamLib/mnParamLib.typ, Logical/Mewa/KGFramework/Pkg_mnParam/mnParamLib/mnParamLib.var, Logical/Mewa/KGFramework/Pkg_mnParam/mnParamLib/mnParamLib.fun, Logical/Mewa/KGFramework/Pkg_mnParam/mnParamLib/mnParam_BinarySearchInNumeric.st, Logical/Mewa/KGFramework/Pkg_mnParam/mnParamLib/mnParam_BinarySearchInString.st, Logical/Mewa/KGFramework/Pkg_mnParam/mnParamLib/mnParam_CountLines.st, Logical/Mewa/KGFramework/Pkg_mnParam/mnParamLib/mnParam_GetCsvDat.st, Logical/Mewa/KGFramework/Pkg_mnParam/mnParamLib/mnParam_atodatetime.st, Logical/Mewa/KGFramework/Pkg_mnParam/mnParamLib/mnParam_GetNextSubstring.st, Logical/Mewa/KGFramework/Pkg_mnParam/mnParamLib/mnParam_GetContainerOfParamNum.st, Logical/Mewa/KGFramework/Pkg_mnParam/mnParamLib/mnParam_GetContainerOfParamStrin.st, Logical/Mewa/KGFramework/Pkg_mnParam/mnParamLib/GetArrayPV.st, Logical/Mewa/KGFramework/Pkg_mnParam/mnParamLib/mnParam_WritePVNum.st, Logical/Mewa/KGFramework/Pkg_mnParam/mnParamLib/mnParam_WritePVrNum.st, Logical/Mewa/KGFramework/Pkg_mnParam/mnParamLib/mnParam_WritePVString.st, Logical/Mewa/KGFramework/Pkg_mnParam/mnParamLib/mnParam_WriteBOM_Mem.st, Logical/Mewa/KGFramework/Pkg_mnParam/mnParamLib/mnParam_WriteNewline_Mem.st, Logical/Mewa/KGFramework/Pkg_mnParam/mnParamLib/mnParam_WriteCSV10_Mem.st, Logical/Mewa/KGFramework/Pkg_mnParam/mnParamLib/mnParam_WriteCSV11_Mem.st, Logical/Mewa/KGFramework/Pkg_mnParam/mnParamLib/mnParam_WriteCSV20_Mem.st, Logical/Mewa/KGFramework/Pkg_mnParam/mnParamLib/mnParam_WriteCSV81_Mem.st, Logical/Mewa/KGFramework/Pkg_mnParam/mnParamLib/mnParam_WriteCSV80_Mem.st, Logical/Mewa/KGFramework/Pkg_mnParam/mnParamLib/mnParam_WriteCSV90_Mem.st, Logical/Mewa/KGFramework/Pkg_mnParam/mnParamLib/mnParam_WriteCSV251_Mem.st, Logical/Mewa/KGFramework/Pkg_mnParam/mnParamLib/mnParam_WriteCSV252_Mem.st, Logical/Mewa/KGFramework/Pkg_mnParam/mnParamLib/mnParam_WriteCSV253_Mem.st, Logical/Mewa/KGFramework/Pkg_mnParam/mnParamLib/mnParam_WriteCSV254_Mem.st, Logical/Mewa/KGFramework/Pkg_mnParam/mnParamLib/mnParam_WriteCSV255_Mem.st, Logical/Mewa/KGFramework/Pkg_mnParam/mnParamLib/mnParam_datetimetoa.st, Logical/Mewa/KGFramework/Pkg_mnParam/mnParamLib/mnParam_datetoa.st, Logical/Mewa/KGFramework/Pkg_mnTxt/Pkg_mnTxt.typ, Logical/Mewa/KGFramework/Pkg_mnTxt/Pkg_mnTxt.var, Logical/Mewa/KGFramework/Pkg_mnTxt/mnTxt/mnTxt.typ, Logical/Mewa/KGFramework/Pkg_hlDFII/Pkg_hlDFII.var, Logical/Mewa/KGFramework/Pkg_hlKanLink/hlKanLink.typ, Logical/Mewa/KGFramework/Pkg_hlKanLink/hlKanLink/KL_SaveConfDO.st, Logical/Mewa/KGFramework/Pkg_hlKanLink/hlKanLink/KanLink.fun, Logical/Mewa/KGFramework/Pkg_hlKanLink/KanLinkLib/KLLib_InitCltPV.st, Logical/Mewa/KGFramework/Pkg_mnTest/Pkg_mnTest.typ, Logical/Mewa/KGFramework/Pkg_mnTest/mnTest/mnTestInit.st, Logical/Mewa/KGFramework/Pkg_mnTest/mnTest/mnTestExit.st, Logical/Mewa/KGFramework/Pkg_mnTest/mnTest/mnTest.typ, Logical/Mewa/KGFramework/Pkg_svCPCache/svCPCache/svCPCacheExit.st, Logical/Mewa/KGFramework/Pkg_svCPCache/svCPCache/_actFillCPList.st, Logical/Mewa/KGFramework/Pkg_svCPCache/svCPCache/svCPCache.fun, Logical/Mewa/KGFrameworkShare/mnCntGlob.var, Logical/Mewa/KGFrameworkShare/mnTxtGlob.var, Logical/Mewa/KGFrameworkShare/mnParamGlob.var, Logical/Mewa/KGFrameworkShare/svCPCacheGlob.var, Logical/Mewa/KGFrameworkShare/Pkg_KGStandardShare/KGStandardShare.kgMsgStatus.var, Logical/Mewa/KGFrameworkShare/Pkg_KGStandardShare/kgdevice.var, Logical/Mewa/KGFrameworkShare/Pkg_mnEthShare/Pkg_mnEthShare.var, Logical/Mewa/KGFrameworkShare/Pkg_mnMsgShare/Pkg_mnMsgShare.var, Logical/Mewa/KGFrameworkShare/Pkg_hlKanLinkUser/Pkg_hlKanLinkUser.var, Logical/Mewa/KGFrameworkShare/Pkg_hlKanLinkUser/KL_UserLib/Batch.typ, Logical/Mewa/KGFrameworkShare/Pkg_hlKanLinkUser/KL_UserLib/KL_UserLib.typ, Logical/Mewa/KGFrameworkShare/Pkg_hlKanLinkUser/KL_UserLib/KL_OnRecReq.st, Logical/Mewa/KGFrameworkShare/Pkg_hlKanLinkUser/KL_UserLib/KL_UserLib.fun, Logical/Mewa/KGFrameworkShare/Pkg_hlKanLinkUser/KL_UserLib/CmdWetExt.typ, Logical/Mewa/KGFrameworkShare/Pkg_mnTestUser/libTestUse/libTest.typ, Logical/Mewa/KGFrameworkShare/Pkg_mnTestUser/libTestUse/libTestUse.typ, Logical/Mewa/KGFrameworkShare/Pkg_mnTestUser/libTestUse/libTest.var, Logical/Mewa/KGFrameworkShare/Pkg_mnTestUser/libTestUse/libTestUse.var, Logical/Mewa/KGFrameworkShare/Pkg_mnTestUser/libTestUse/TestUser_StopTask.st, Logical/Mewa/KGFrameworkShare/Pkg_mnTestUser/libTestUse/TestUser_SetMode.st, Logical/Mewa/KGFrameworkShare/Pkg_mnTestUser/libTestUse/TestUser_RunTest.st, Logical/Mewa/KGFrameworkShare/Pkg_mnTestUser/libTestUse/libTestUse.fun, Logical/Mewa/KGFrameworkShare/Pkg_mnTestUser/mnTestUser/mnTestUserCyclic.st, Logical/Mewa/KGFrameworkShare/Pkg_mnTestUser/mnTestUser/mnTestUserInit.st, Logical/Mewa/KGFrameworkShare/Pkg_mnTestUser/mnTestUser/mnTestUserExit.st, Logical/Mewa/KGFrameworkShare/Pkg_mnTestUser/mnTestUser/mnTestUser.typ, Logical/Mewa/KGFrameworkShare/Pkg_mnTestUser/mnTestUser/mnTestUser.var
